PROGRAM AlarmExtension
VAR
	bAlarmi			: BOOL;
	iAlarm			: INT;
	eState			: E_STATE;
	
	bToggleState	: BOOL;
END_VAR

IF bToggleState THEN
	bToggleState := FALSE;
	IF eState = E_STATE.normal THEN
		eState := E_STATE.error;
	ELSE
		eState := E_STATE.normal;	
	END_IF
END_IF

END_PROGRAM

(* stored: Version 1.1.0.1, ProductVersion 3.1.4024.12
   POU AlarmExtension: Id {71f17bd9-7d63-4186-92a0-ef15b2b9e51e}, SpecialFunc None *)
